// TIA Portal V20 export
TYPE "sAxis_CMD"
   STRUCT
      bEnableAxis : Bool;   // 使能
      bResetAxis : Bool;   // 复位
      bjogForward : Bool;   // Taster Aufwärts / 正点
      bjogBackward : Bool;   // Taster Abwärts / 反点
      bmoveVelocity : Bool;   // 速度运行
      bstop : Bool;   // 停止
      bfastStop : Bool;   // 急停
      bHoming : Bool;   // 回零
      bGoToPos : Array[0..16] of Bool;   // Start Aufwärts in Automatik / 16个定位
      iGoToPos : Word;   // 16个定位 Word
      bCallAbsPos : Bool;   // 定位位置切换时，单独的定位按钮
      bRelPos : Bool;   // 相对定位
      MyBool : Array[0..5] of Bool;   // 临时变量
   END_STRUCT;
END_TYPE
